FUNCTION_BLOCK Mailbox
  (* Version 1.0, 2006-11-02, Goran Cengic, Chalmers *)
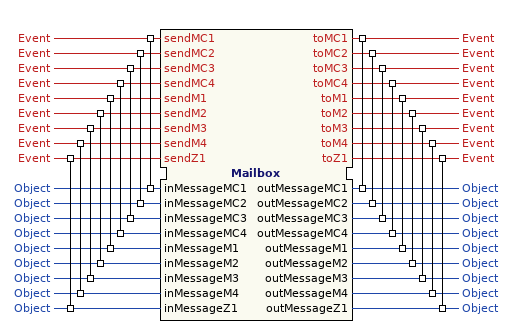
  EVENT_INPUT
    sendMC1 WITH inMessageMC1;
    sendMC2 WITH inMessageMC2;
    sendMC3 WITH inMessageMC3;
    sendMC4 WITH inMessageMC4;
    sendM1 WITH inMessageM1;
    sendM2 WITH inMessageM2;
    sendM3 WITH inMessageM3;
    sendM4 WITH inMessageM4;
    sendZ1 WITH inMessageZ1;
  END_EVENT
  EVENT_OUTPUT
    toMC1 WITH outMessageMC1;
    toMC2 WITH outMessageMC2;
    toMC3 WITH outMessageMC3;
    toMC4 WITH outMessageMC4;
    toM1 WITH outMessageM1;
    toM2 WITH outMessageM2;
    toM3 WITH outMessageM3;
    toM4 WITH outMessageM4;
    toZ1 WITH outMessageZ1;
  END_EVENT
  VAR_INPUT
    inMessageMC1 : Object;
    inMessageMC2 : Object;
    inMessageMC3 : Object;
    inMessageMC4 : Object;
    inMessageM1 : Object;
    inMessageM2 : Object;
    inMessageM3 : Object;
    inMessageM4 : Object;
    inMessageZ1 : Object;
  END_VAR
  VAR_OUTPUT
    outMessageMC1 : Object;
    outMessageMC2 : Object;
    outMessageMC3 : Object;
    outMessageMC4 : Object;
    outMessageM1 : Object;
    outMessageM2 : Object;
    outMessageM3 : Object;
    outMessageM4 : Object;
    outMessageZ1 : Object;
  END_VAR
END_FUNCTION_BLOCK
